FUNCTION BandPassFilter : REAL
VAR_INPUT
	Error : REAL;
	
	BPF : POINTER TO BandPassFilterStruct;
	
	Enable : BOOL;
	
END_VAR
VAR
END_VAR

BandPassFilter := BPF^.G1_b0*(Error - BPF^.error2) - BPF^.output1*BPF^.G1_a1 - BPF^.output2*BPF^.G1_a2;

IF Enable = TRUE THEN
	BPF^.error1 := Error;
	BPF^.error2 := BPF^.error1;
	BPF^.output1 := BandPassFilter;
	BPF^.output2 := BPF^.output1;
ELSE
	BPF^.error1 := 0;
	BPF^.error2 := 0;
	BPF^.output1 := 0;
	BPF^.output2 := 0;
	BandPassFilter := 0;
END_IF

END_FUNCTION

(* stored: Version 1.1.0.1, ProductVersion 3.1.4024.4
   POU BandPassFilter: Id {4133bbff-f006-4144-835a-edde2dcf8487}, SpecialFunc None *)
